SUBAPPLICATION Abscheider (* Subapplication Type *)
  (* Standard: 61499-2 *)
  (* Version 1.0, 2023-01-29, Franz *)
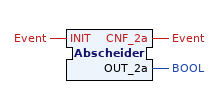
  EVENT_INPUT
    INIT;
  END_EVENT
  EVENT_OUTPUT
    CNF_2a;
  END_EVENT
  VAR_OUTPUT
    OUT_2a : BOOL;
  END_VAR
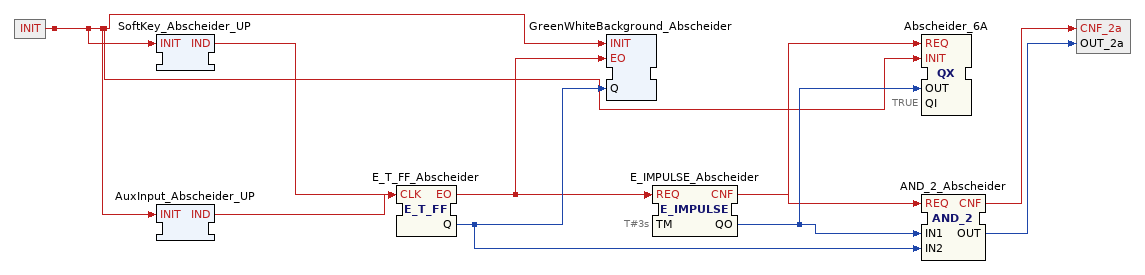
  FBS
    AND_2_Abscheider : AND_2;
    E_T_FF_Abscheider : E_T_FF;
    Abscheider_6A : QX(QI := TRUE);
    E_IMPULSE_Abscheider : E_IMPULSE(TM := T#3s);
  END_FBS
  SUBAPPLICATION AuxInput_Abscheider_UP
    EVENT_INPUT
      INIT;
    END_EVENT
    EVENT_OUTPUT
      IND;
    END_EVENT
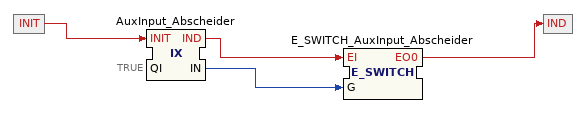
    FBS
      E_SWITCH_AuxInput_Abscheider : E_SWITCH;
      AuxInput_Abscheider : IX(QI := TRUE);
    END_FBS
    EVENT_CONNECTIONS
      AuxInput_Abscheider.IND TO E_SWITCH_AuxInput_Abscheider.EI;
      INIT TO AuxInput_Abscheider.INIT;
      E_SWITCH_AuxInput_Abscheider.EO0 TO IND;
    END_CONNECTIONS
    DATA_CONNECTIONS
      AuxInput_Abscheider.IN TO E_SWITCH_AuxInput_Abscheider.G;
    END_CONNECTIONS
  END_SUBAPPLICATION
  SUBAPPLICATION SoftKey_Abscheider_UP
    EVENT_INPUT
      INIT;
    END_EVENT
    EVENT_OUTPUT
      IND;
    END_EVENT
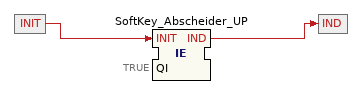
    FBS
      SoftKey_Abscheider_UP : IE(QI := TRUE);
    END_FBS
    EVENT_CONNECTIONS
      INIT TO SoftKey_Abscheider_UP.INIT;
      SoftKey_Abscheider_UP.IND TO IND;
    END_CONNECTIONS
  END_SUBAPPLICATION
  SUBAPPLICATION GreenWhiteBackground_Abscheider
    EVENT_INPUT
      INIT;
      EO;
    END_EVENT
    VAR_INPUT
      Q : BOOL;
    END_VAR
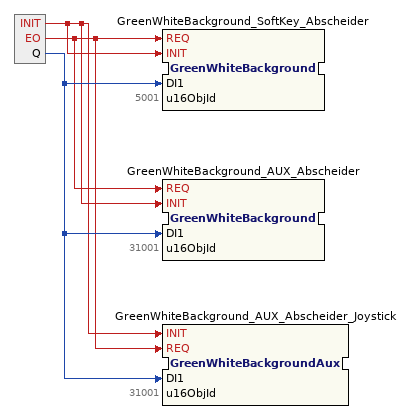
    FBS
      GreenWhiteBackground_SoftKey_Abscheider : GreenWhiteBackground(u16ObjId := 5001);
      GreenWhiteBackground_AUX_Abscheider : GreenWhiteBackground(u16ObjId := 31001);
      GreenWhiteBackground_AUX_Abscheider_Joystick : GreenWhiteBackgroundAux(u16ObjId := 31001);
    END_FBS
    EVENT_CONNECTIONS
      EO TO GreenWhiteBackground_SoftKey_Abscheider.REQ;
      INIT TO GreenWhiteBackground_SoftKey_Abscheider.INIT;
      EO TO GreenWhiteBackground_AUX_Abscheider.REQ;
      INIT TO GreenWhiteBackground_AUX_Abscheider.INIT;
      INIT TO GreenWhiteBackground_AUX_Abscheider_Joystick.INIT;
      EO TO GreenWhiteBackground_AUX_Abscheider_Joystick.REQ;
    END_CONNECTIONS
    DATA_CONNECTIONS
      Q TO GreenWhiteBackground_SoftKey_Abscheider.DI1;
      Q TO GreenWhiteBackground_AUX_Abscheider.DI1;
      Q TO GreenWhiteBackground_AUX_Abscheider_Joystick.DI1;
    END_CONNECTIONS
  END_SUBAPPLICATION
  EVENT_CONNECTIONS
    E_IMPULSE_Abscheider.CNF TO AND_2_Abscheider.REQ;
    E_T_FF_Abscheider.EO TO E_IMPULSE_Abscheider.REQ;
    E_IMPULSE_Abscheider.CNF TO Abscheider_6A.REQ;
    AND_2_Abscheider.CNF TO CNF_2a;
    INIT TO SoftKey_Abscheider_UP.INIT;
    SoftKey_Abscheider_UP.IND TO E_T_FF_Abscheider.CLK;
    INIT TO AuxInput_Abscheider_UP.INIT;
    AuxInput_Abscheider_UP.IND TO E_T_FF_Abscheider.CLK;
    INIT TO Abscheider_6A.INIT;
    INIT TO GreenWhiteBackground_Abscheider.INIT;
    E_T_FF_Abscheider.EO TO GreenWhiteBackground_Abscheider.EO;
  END_CONNECTIONS
  DATA_CONNECTIONS
    E_IMPULSE_Abscheider.QO TO AND_2_Abscheider.IN1;
    E_T_FF_Abscheider.Q TO AND_2_Abscheider.IN2;
    E_IMPULSE_Abscheider.QO TO Abscheider_6A.OUT;
    AND_2_Abscheider.OUT TO OUT_2a;
    E_T_FF_Abscheider.Q TO GreenWhiteBackground_Abscheider.Q;
  END_CONNECTIONS
END_SUBAPPLICATION
